// TwinCAT 3 PLC project lamp_motion
// Title: tmo_lamp_motion
// Company: SLAC
// ProjectVersion: 0.0.0
// ProgramVersion: 3.1.4022.7
// libraries:
//   LCLS General, * (SLAC)
//   lcls-twincat-motion, * (SLAC)
//   Tc2_MC2, * (Beckhoff Automation GmbH)
//   Tc2_Standard, * (Beckhoff Automation GmbH)
//   Tc2_System, * (Beckhoff Automation GmbH)
//   Tc2_Utilities, * (Beckhoff Automation GmbH)
//   Tc3_Module, * (Beckhoff Automation GmbH)
// project tree:
//   GVLs/ GVL_PLC_Interfaces.TcGVL
//   / PlcTask.TcTTO
//   POUs/ Main.TcPOU
// real-time tasks:
//   TASK PlcTask: cycle T#9ms, priority 20, ADS port 350
// motion (NC):
//   TASK NC-Task 1 SAF: cycle T#2ms, priority 4, ADS port 501
//   TASK NC-Task 1 SVB: cycle T#10ms, priority 8, ADS port 511
//   AXIS GasJetX (id 1)
//     Dynamic: Acceleration=2, Deceleration=2, DelayTime=0.008
//     Velo: SlowManual=0.5, FastManual=1, Maximum=1
//     OtherSettings: AllowMotionCmdToSlave=true
//     encoder EncType=19
//       EncPara: ScaleFactorNumerator=5e-05, Inverse=true, MaxCount=#xffffffff
//         SoftEndMinControl: Range=-2
//         SoftEndMaxControl: Range=2
//         Inc: RefSoftSyncMask=#x0000ffff
//     drive DrvType=24
//       DrvPara: Inverse=true
//         Analog: VeloReferenz=12.7, ScaleFactorActTorque=0.1
//         TimeComp: TaskDelayCycles=1
//     controller CtrType=1
//       CtrPara: PriorControlFactor=1
//         PosDiffControl: Range=0.8
//         Observer: BandWidth=20
//   AXIS GasJetY (id 2)
//     Dynamic: Acceleration=2, Deceleration=2, DelayTime=0.008
//     Velo: RefSearch=1, RefSync=1, SlowManual=0.5, FastManual=1, Maximum=8
//     OtherSettings: AllowMotionCmdToSlave=true
//     encoder EncType=19
//       EncPara: ScaleFactorNumerator=5e-05, MaxCount=#xffffffff
//         SoftEndMaxControl: Enable=true, Range=735
//         Inc: RefSoftSyncMask=#x0000ffff
//     drive DrvType=24
//       Analog: VeloReferenz=10, ScaleFactorActTorque=0.1
//       TimeComp: TaskDelayCycles=1
//     controller CtrType=1
//       CtrPara: PriorControlFactor=1
//         PosDiffControl: Range=0.8
//         PID: PosKp=2
//         Observer: BandWidth=20
//   AXIS GasJetZ (id 3)
//     Dynamic: AccelerationMaximum=130, DecelerationMaximum=130, Acceleration=3.01464, Deceleration=3.01464, Jerk=17.8197, DelayTime=0.008
//     Velo: SlowManual=0.5, FastManual=1, Maximum=1
//     TargetPosControl: Range=0.01
//     OtherSettings: AllowMotionCmdToSlave=true
//     encoder EncType=29
//       EncPara: ScaleFactorNumerator=5e-05, MaxCount=#xffffffff
//         Inc: RefSoftSyncMask=#x0000ffff
//     drive DrvType=24
//       DrvPara: Inverse=true
//         Analog: VeloReferenz=12.7, ScaleFactorActTorque=0.1
//         TimeComp: TaskDelayCycles=1
//     controller CtrType=1
//       CtrPara: PriorControlFactor=1
//         PosDiffControl: Range=0.1, Time=0.1
//         Observer: BandWidth=20
//   AXIS GasNeedleX (id 4)
//     Dynamic: Acceleration=0.5, Deceleration=2, DelayTime=0.008
//     Velo: SlowManual=0.5, FastManual=1, Maximum=1
//     PositionAreaControl: Range=0.005
//     OtherSettings: AllowMotionCmdToSlave=true
//     encoder EncType=29
//       EncPara: ScaleFactorNumerator=5e-05, Offset=-214613, MaxCount=#xffffffff
//         SoftEndMinControl: Enable=true, Range=19
//         SoftEndMaxControl: Enable=true, Range=39.5
//         Inc: RefSoftSyncMask=#x0000ffff
//     drive DrvType=24
//       Analog: VeloReferenz=10, ScaleFactorActTorque=0.1
//       TimeComp: TaskDelayCycles=1
//     controller CtrType=1
//       CtrPara: PriorControlFactor=1
//         PosDiffControl: Range=0.5
//         PID: PosKp=2
//         Observer: BandWidth=20
//   AXIS GasNeedleY (id 5)
//     Dynamic: Acceleration=2, Deceleration=2, DelayTime=0.008
//     Velo: SlowManual=0.5, FastManual=1, Maximum=1
//     PositionAreaControl: Range=0.5
//     TargetPosControl: Range=0.001, Time=0.2
//     OtherSettings: AllowMotionCmdToSlave=true
//     encoder EncType=19
//       EncPara: ScaleFactorNumerator=5e-05, MaxCount=#xffffffff
//         Inc: RefSoftSyncMask=#x0000ffff
//     drive DrvType=24
//       Analog: VeloReferenz=13, ScaleFactorActTorque=0.1
//       TimeComp: TaskDelayCycles=1
//     controller CtrType=1
//       CtrPara: PriorControlFactor=1
//         PosDiffControl: Range=0.5
//         PID: PosKp=5
//         Observer: BandWidth=20
//   AXIS GasNeedleZ (id 6)
//     Dynamic: Acceleration=2, Deceleration=2, DelayTime=0.008
//     Velo: SlowManual=0.5, FastManual=1, Maximum=1
//     PositionAreaControl: Range=0.005
//     TargetPosControl: Range=0.5
//     OtherSettings: AllowMotionCmdToSlave=true
//     encoder EncType=19
//       EncPara: ScaleFactorNumerator=5e-05, Inverse=true, MaxCount=#xffffffff
//         SoftEndMinControl: Enable=true, Range=-50
//         SoftEndMaxControl: Enable=true, Range=-25
//         Inc: RefSoftSyncMask=#x0000ffff
//     drive DrvType=24
//       Analog: VeloReferenz=10.5, ScaleFactorActTorque=0.1
//       TimeComp: TaskDelayCycles=1
//     controller CtrType=1
//       CtrPara: PriorControlFactor=1
//         PosDiffControl: Range=0.5
//         Observer: BandWidth=20
//   AXIS SamplePaddleX (id 7)
//     Dynamic: Acceleration=2, Deceleration=2, DelayTime=0.008
//     Velo: Maximum=1
//     TargetPosControl: Range=0.001, Time=0.1
//     OtherSettings: AllowMotionCmdToSlave=true
//     encoder EncType=4
//       EncPara: ScaleFactorNumerator=1e-05, Inverse=true, MaxCount=#xffffffff
//         SoftEndMinControl: Range=-39
//         Inc: RefSoftSyncMask=#x0000ffff
//     drive DrvType=24
//       DrvPara: Inverse=true
//         Analog: VeloReferenz=10, ScaleFactorActTorque=0.1
//         TimeComp: TaskDelayCycles=1
//     controller CtrType=2
//       CtrPara: PriorControlFactor=1
//         PosDiffControl: Range=1
//         PID: PosKp=20, PosExtKp=50, DeadBandPosition=0.0005
//         Observer: BandWidth=20
//   AXIS SamplePaddleY (id 8)
//     Dynamic: Acceleration=2, Deceleration=2, DelayTime=0.008
//     Velo: Maximum=1
//     TargetPosControl: Range=0.001, Time=0.1
//     OtherSettings: AllowMotionCmdToSlave=true
//     encoder EncType=4
//       EncPara: ScaleFactorNumerator=2e-05, Inverse=true, MaxCount=#xffffffff
//         SoftEndMinControl: Range=-10
//         SoftEndMaxControl: Range=10
//         Inc: RefSoftSyncMask=#x0000ffff
//     drive DrvType=24
//       DrvPara: Inverse=true
//         Analog: VeloReferenz=5, ScaleFactorActTorque=0.1
//         TimeComp: TaskDelayCycles=1
//     controller CtrType=2
//       CtrPara: PriorControlFactor=1
//         PosDiffControl: Range=0.5
//         PID: PosKp=20, PosExtKp=50, DeadBandPosition=0.0005
//         Observer: BandWidth=20
//   AXIS SamplePaddleZ (id 9)
//     Dynamic: Acceleration=2, Deceleration=2, DelayTime=0.008
//     Velo: Maximum=1
//     TargetPosControl: Range=0.001, Time=0.1
//     OtherSettings: AllowMotionCmdToSlave=true
//     encoder EncType=4
//       EncPara: ScaleFactorNumerator=1e-05, Inverse=true, MaxCount=#xffffffff
//         Inc: RefSoftSyncMask=#x0000ffff
//     drive DrvType=24
//       DrvPara: Inverse=true
//         Analog: VeloReferenz=10, ScaleFactorActTorque=0.1
//         TimeComp: TaskDelayCycles=1
//     controller CtrType=2
//       CtrPara: PriorControlFactor=1
//         PosDiffControl: Range=1
//         PID: PosKp=20, PosExtKp=50, DeadBandPosition=0.0005
//         Observer: BandWidth=20
//   AXIS FlowCellX (id 10)
//     Dynamic: Acceleration=2, Deceleration=2
//     Velo: Maximum=1
//     OtherSettings: AllowMotionCmdToSlave=true
//     encoder EncType=1
//       EncPara: ScaleFactorNumerator=9.375e-05, ScaleFactorDenominator=1.2
//         Inc: RefSoftSyncMask=#x0000ffff
//     drive DrvType=5
//       Analog: VeloReferenz=10, ScaleFactorActTorque=0.1
//       TimeComp: TaskDelayCycles=1
//     controller CtrType=1
//       CtrPara: PriorControlFactor=1
//         PosDiffControl: Range=0.5
//         Observer: BandWidth=20
//   AXIS FlowCellY (id 11)
//     Dynamic: Acceleration=2, Deceleration=2
//     Velo: Maximum=1
//     OtherSettings: AllowMotionCmdToSlave=true
//     encoder EncType=1
//       EncPara: ScaleFactorNumerator=7.8125e-05, ScaleFactorDenominator=0.8
//         Inc: RefSoftSyncMask=#x0000ffff
//     drive DrvType=5
//       Analog: VeloReferenz=12.5, ScaleFactorActTorque=0.1
//       TimeComp: TaskDelayCycles=1
//     controller CtrType=1
//       CtrPara: PriorControlFactor=1
//         PosDiffControl: Range=0.5
//         Observer: BandWidth=20
//   AXIS FlowCellZ (id 12)
//     Dynamic: Acceleration=2, Deceleration=2
//     Velo: Maximum=1
//     OtherSettings: AllowMotionCmdToSlave=true
//     encoder EncType=1
//       EncPara: ScaleFactorNumerator=7.8125e-05
//         Inc: RefSoftSyncMask=#x0000ffff
//     drive DrvType=5
//       Analog: VeloReferenz=10, ScaleFactorActTorque=0.1
//       TimeComp: TaskDelayCycles=1
//     controller CtrType=1
//       CtrPara: PriorControlFactor=1
//         PosDiffControl: Range=0.5
//         Observer: BandWidth=20
//   AXIS FlowCellTheta (id 13)
//     General: UnitName=Degree
//     Velo: Maximum=10
//     OtherSettings: AllowMotionCmdToSlave=true
//     encoder EncType=1
//       EncPara: ScaleFactorNumerator=0.0003125
//         Inc: RefSoftSyncMask=#x0000ffff
//     drive DrvType=5
//       Analog: VeloReferenz=40, ScaleFactorActTorque=0.1
//       TimeComp: TaskDelayCycles=1
//     controller CtrType=2
//       CtrPara: PriorControlFactor=1
//         PosDiffControl: Range=0.5
//         Observer: BandWidth=20
//   AXIS TIXELX (id 14)
//     Dynamic: Acceleration=2, Deceleration=2, DelayTime=0.008
//     Velo: Maximum=1
//     OtherSettings: AllowMotionCmdToSlave=true
//     encoder EncType=4
//       EncPara: ScaleFactorNumerator=3.90625e-05, Inverse=true, MaxCount=#x0000ffff
//         SoftEndMinControl: Range=-2
//         SoftEndMaxControl: Range=2
//         Inc: RefSoftSyncMask=#x0000ffff
//     drive DrvType=24
//       DrvPara: Inverse=true
//         Analog: VeloReferenz=5, ScaleFactorActTorque=0.1
//         TimeComp: TaskDelayCycles=1
//     controller CtrType=1
//       CtrPara: PriorControlFactor=1
//         PosDiffControl: Range=0.5
//         Observer: BandWidth=20
//   AXIS TIXELY (id 15)
//     Dynamic: Acceleration=2, Deceleration=2, DelayTime=0.008
//     Velo: Maximum=1
//     OtherSettings: AllowMotionCmdToSlave=true
//     encoder EncType=4
//       EncPara: ScaleFactorNumerator=3.90625e-05, Inverse=true, MaxCount=#x0000ffff
//         SoftEndMinControl: Range=-2
//         SoftEndMaxControl: Range=2
//         Inc: RefSoftSyncMask=#x0000ffff
//     drive DrvType=24
//       DrvPara: Inverse=true
//         Analog: VeloReferenz=5, ScaleFactorActTorque=0.1
//         TimeComp: TaskDelayCycles=1
//     controller CtrType=1
//       CtrPara: PriorControlFactor=1
//         PosDiffControl: Range=0.5
//         Observer: BandWidth=20
//   AXIS TIXELZ (id 16)
//     Dynamic: Acceleration=2, Deceleration=2, DelayTime=0.008
//     Velo: Maximum=1
//     OtherSettings: AllowMotionCmdToSlave=true
//     encoder EncType=4
//       EncPara: ScaleFactorNumerator=3.90625e-05, Inverse=true, MaxCount=#x0000ffff
//         SoftEndMinControl: Range=-2
//         SoftEndMaxControl: Range=2
//         Inc: RefSoftSyncMask=#x0000ffff
//     drive DrvType=24
//       DrvPara: Inverse=true
//         Analog: VeloReferenz=5, ScaleFactorActTorque=0.1
//         TimeComp: TaskDelayCycles=1
//     controller CtrType=1
//       CtrPara: PriorControlFactor=1
//         PosDiffControl: Range=0.5
//         Observer: BandWidth=20
// I/O:
//   DEVICE PLC Rail (EtherCAT), AmsNetId 0.0.0.0.2.1
//     Power (EK1200) [EK1200-5000 EtherCAT Power supply (2A E-Bus)]
//       PMPS_FFO [EL2202 2Ch. Dig. Output 24V, 0.5A]
//       License (EL6070) [EL6070 1Ch. Licensing-Terminal]
//       LAMP_MOTION_E03_EL6695 [EL6695 EtherCAT Bridge terminal (Primary)]
//       PLC Junction 1 (EK1122) [EK1122 2 port EtherCAT junction]
//         X1 AtmosphereMotion (EK1100) [EK1100 EtherCAT Coupler (2A E-Bus)]
//           GasJetX-EL7041 [EL7041 1Ch. Stepper motor output stage (50V, 5A)]
//           GasJetY-EL7041 [EL7041 1Ch. Stepper motor output stage (50V, 5A)]
//           GasJetY-Brake-EL2004 [EL2004 4Ch. Dig. Output 24V, 0.5A]
//           GasJetZ-EL7041 [EL7041 1Ch. Stepper motor output stage (50V, 5A)]
//           GasNeedleX-EL7041 [EL7041 1Ch. Stepper motor output stage (50V, 5A)]
//           GasNeedleY-EL7041 [EL7041 1Ch. Stepper motor output stage (50V, 5A)]
//           GasNeedleZ-EL7041 [EL7041 1Ch. Stepper motor output stage (50V, 5A)]
//           FlowCellTheta-EL7041 [EL7041 1Ch. Stepper motor output stage (50V, 5A)]
//           GasJetXY-EL5042 [EL5042 2Ch. BiSS-C Encoder]
//           GasJetZGasNeedleX-EL5042 [EL5042 2Ch. BiSS-C Encoder]
//           GasNeedleYZ-EL5042 [EL5042 2Ch. BiSS-C Encoder]
//           AtmosphereMotion-EK1110 [EK1110 EtherCAT extension]
//         X1 VacuumMotion (EK1100) [EK1100 EtherCAT Coupler (2A E-Bus)]
//           SamplePaddleX-EL7041 [EL7041 1Ch. Stepper motor output stage (50V, 5A)]
//           SamplePaddleXY-EL1084 [EL1084 4Ch. Dig. Input 24V, 3ms, negative]
//           SamplePaddleY-EL7041 [EL7041 1Ch. Stepper motor output stage (50V, 5A)]
//           SamplePaddleX-EL5021 [EL5021 1Ch. Sin/Cos Encoder]
//           SamplePaddleY-EL5021 [EL5021 1Ch. Sin/Cos Encoder]
//           SamplePaddleZ-EL7041 [EL7041 1Ch. Stepper motor output stage (50V, 5A)]
//           SamplePaddleZ-EL1084 [EL1084 4Ch. Dig. Input 24V, 3ms, negative]
//           SamplePaddleZ-EL5021 [EL5021 1Ch. Sin/Cos Encoder]
//           Term 56 (EL9410) [EL9410 E-Bus Power Supplier  (Diagnostics)]
//           Term 57 (EL7041) [EL7041 1Ch. Stepper motor output stage (50V, 5A)]
//           Term 58 (EL5021) [EL5021 1K. Sin/Cos Encoder]
//           Term 59 (EL1084) [EL1084 4Ch. Dig. Input 24V, 3ms, negative]
//           Term 60 (EL7041) [EL7041 1Ch. Stepper motor output stage (50V, 5A)] (disabled)
//           Term 61 (EL5021) [EL5021 1Ch. Sin/Cos Encoder]
//           Term 69 (EL9011) [EL9011 End Terminal]
//         TIXEL (EK1100) [EK1100 EtherCAT Coupler (2A E-Bus)]
//           TIXELX-EL7041 [EL7041 1Ch. Stepper motor output stage (50V, 5A)]
//           TIXELXY_ENC-EL5042 [EL5042 2Ch. BiSS-C Encoder]
//           TIXELY-EL7041 [EL7041 1Ch. Stepper motor output stage (50V, 5A)]
//           TIXELZ-EL7041 [EL7041 1Ch. Stepper motor output stage (50V, 5A)]
//           TIXELZ_ENC-EL5042 [EL5042 2Ch. BiSS-C Encoder]
//           Term 68 (EK1110)
// variable links:
//   (this object) <-> PLC Rail (EtherCAT)/Power (EK1200)/PLC Junction 1 (EK1122)/X1 AtmosphereMotion (EK1100)/GasJetX-EL7041
//     Drive/Inputs/In/nState1 @bit 3 <-> STM Status/Status/Error
//     Drive/Inputs/In/nState1 @bit 5 <-> STM Status/Status/Moving negative
//     Drive/Inputs/In/nState1 @bit 4 <-> STM Status/Status/Moving positive
//     Drive/Inputs/In/nState1 @bit 1 <-> STM Status/Status/Ready
//     Drive/Inputs/In/nState1 <-> STM Status/Status/Ready to enable
//     Drive/Inputs/In/nState1 @bit 6 <-> STM Status/Status/Torque reduced
//     Drive/Inputs/In/nState1 @bit 2 <-> STM Status/Status/Warning
//     Drive/Inputs/In/nState2 @bit 3 <-> STM Status/Status/Digital input 1
//     Drive/Inputs/In/nState2 @bit 4 <-> STM Status/Status/Digital input 2
//     Drive/Inputs/In/nState2 @bit 5 <-> STM Status/Status/Sync error
//     Drive/Inputs/In/nState2 @bit 7 <-> STM Status/Status/TxPDO Toggle
//     Drive/Inputs/In/nState4 @bit 1 <-> WcState/InputToggle
//     Drive/Inputs/In/nState4 <-> WcState/WcState
//     Drive/Outputs/Out/nCtrl1 <-> STM Control/Control/Enable
//     Drive/Outputs/Out/nCtrl1 @bit 2 <-> STM Control/Control/Reduce torque
//     Drive/Outputs/Out/nCtrl1 @bit 1 <-> STM Control/Control/Reset
//     Drive/Outputs/Out/nDataOut2[0] <-> STM Velocity/Velocity
//   (this object) <-> PLC Rail (EtherCAT)/Power (EK1200)/PLC Junction 1 (EK1122)/X1 AtmosphereMotion (EK1100)/GasJetXY-EL5042
//     Enc/Inputs/In/nDataIn1 <-> FB Inputs Channel 1 compact/Position
//     Enc/Inputs/In/nDataIn1 <-> FB Inputs Channel 2 compact/Position
//     Enc/Inputs/In/nState1 @bit 1 <-> FB Inputs Channel 1 compact/Status/Error
//     Enc/Inputs/In/nState1 @bit 1 <-> FB Inputs Channel 2 compact/Status/Error
//     Enc/Inputs/In/nState1 @bit 2 <-> FB Inputs Channel 1 compact/Status/Ready
//     Enc/Inputs/In/nState1 @bit 2 <-> FB Inputs Channel 2 compact/Status/Ready
//     Enc/Inputs/In/nState1 <-> FB Inputs Channel 1 compact/Status/Warning
//     Enc/Inputs/In/nState1 <-> FB Inputs Channel 2 compact/Status/Warning
//     Enc/Inputs/In/nState2 @bit 4 <-> FB Inputs Channel 1 compact/Status/Diag
//     Enc/Inputs/In/nState2 @bit 4 <-> FB Inputs Channel 2 compact/Status/Diag
//     Enc/Inputs/In/nState2 @bit 6 <-> FB Inputs Channel 1 compact/Status/Input cycle counter
//     Enc/Inputs/In/nState2 @bit 6 <-> FB Inputs Channel 2 compact/Status/Input cycle counter
//     Enc/Inputs/In/nState2 @bit 5 <-> FB Inputs Channel 1 compact/Status/TxPDO State
//     Enc/Inputs/In/nState2 @bit 5 <-> FB Inputs Channel 2 compact/Status/TxPDO State
//     Enc/Inputs/In/nState4 @bit 1 <-> WcState/InputToggle
//     Enc/Inputs/In/nState4 <-> WcState/WcState
//   (this object) <-> PLC Rail (EtherCAT)/Power (EK1200)/PLC Junction 1 (EK1122)/X1 AtmosphereMotion (EK1100)/GasJetY-EL7041
//     Drive/Inputs/In/nState1 @bit 3 <-> STM Status/Status/Error
//     Drive/Inputs/In/nState1 @bit 5 <-> STM Status/Status/Moving negative
//     Drive/Inputs/In/nState1 @bit 4 <-> STM Status/Status/Moving positive
//     Drive/Inputs/In/nState1 @bit 1 <-> STM Status/Status/Ready
//     Drive/Inputs/In/nState1 <-> STM Status/Status/Ready to enable
//     Drive/Inputs/In/nState1 @bit 6 <-> STM Status/Status/Torque reduced
//     Drive/Inputs/In/nState1 @bit 2 <-> STM Status/Status/Warning
//     Drive/Inputs/In/nState2 @bit 3 <-> STM Status/Status/Digital input 1
//     Drive/Inputs/In/nState2 @bit 4 <-> STM Status/Status/Digital input 2
//     Drive/Inputs/In/nState2 @bit 5 <-> STM Status/Status/Sync error
//     Drive/Inputs/In/nState2 @bit 7 <-> STM Status/Status/TxPDO Toggle
//     Drive/Inputs/In/nState4 @bit 1 <-> WcState/InputToggle
//     Drive/Inputs/In/nState4 <-> WcState/WcState
//     Drive/Outputs/Out/nCtrl1 <-> STM Control/Control/Enable
//     Drive/Outputs/Out/nCtrl1 @bit 2 <-> STM Control/Control/Reduce torque
//     Drive/Outputs/Out/nCtrl1 @bit 1 <-> STM Control/Control/Reset
//     Drive/Outputs/Out/nDataOut2[0] <-> STM Velocity/Velocity
//   (this object) <-> PLC Rail (EtherCAT)/Power (EK1200)/PLC Junction 1 (EK1122)/X1 AtmosphereMotion (EK1100)/GasJetZ-EL7041
//     Drive/Inputs/In/nState1 @bit 3 <-> STM Status/Status/Error
//     Drive/Inputs/In/nState1 @bit 5 <-> STM Status/Status/Moving negative
//     Drive/Inputs/In/nState1 @bit 4 <-> STM Status/Status/Moving positive
//     Drive/Inputs/In/nState1 @bit 1 <-> STM Status/Status/Ready
//     Drive/Inputs/In/nState1 <-> STM Status/Status/Ready to enable
//     Drive/Inputs/In/nState1 @bit 6 <-> STM Status/Status/Torque reduced
//     Drive/Inputs/In/nState1 @bit 2 <-> STM Status/Status/Warning
//     Drive/Inputs/In/nState2 @bit 3 <-> STM Status/Status/Digital input 1
//     Drive/Inputs/In/nState2 @bit 4 <-> STM Status/Status/Digital input 2
//     Drive/Inputs/In/nState2 @bit 5 <-> STM Status/Status/Sync error
//     Drive/Inputs/In/nState2 @bit 7 <-> STM Status/Status/TxPDO Toggle
//     Drive/Inputs/In/nState4 @bit 1 <-> WcState/InputToggle
//     Drive/Inputs/In/nState4 <-> WcState/WcState
//     Drive/Outputs/Out/nCtrl1 <-> STM Control/Control/Enable
//     Drive/Outputs/Out/nCtrl1 @bit 2 <-> STM Control/Control/Reduce torque
//     Drive/Outputs/Out/nCtrl1 @bit 1 <-> STM Control/Control/Reset
//     Drive/Outputs/Out/nDataOut2[0] <-> STM Velocity/Velocity
//   (this object) <-> PLC Rail (EtherCAT)/Power (EK1200)/PLC Junction 1 (EK1122)/X1 AtmosphereMotion (EK1100)/GasJetZGasNeedleX-EL5042
//     Enc/Inputs/In/nComState @bit 1 <-> WcState/InputToggle
//     Enc/Inputs/In/nComState <-> WcState/WcState
//     Enc/Inputs/In/nDataIn1 <-> FB Inputs Channel 1/Position
//     Enc/Inputs/In/nDataIn1 <-> FB Inputs Channel 2/Position
//     Enc/Inputs/In/nState1 @bit 12 <-> FB Inputs Channel 1/Status/Diag
//     Enc/Inputs/In/nState1 @bit 12 <-> FB Inputs Channel 2/Status/Diag
//     Enc/Inputs/In/nState1 @bit 1 <-> FB Inputs Channel 1/Status/Error
//     Enc/Inputs/In/nState1 @bit 1 <-> FB Inputs Channel 2/Status/Error
//     Enc/Inputs/In/nState1 @bit 14 <-> FB Inputs Channel 1/Status/Input cycle counter
//     Enc/Inputs/In/nState1 @bit 14 <-> FB Inputs Channel 2/Status/Input cycle counter
//     Enc/Inputs/In/nState1 @bit 2 <-> FB Inputs Channel 1/Status/Ready
//     Enc/Inputs/In/nState1 @bit 2 <-> FB Inputs Channel 2/Status/Ready
//     Enc/Inputs/In/nState1 @bit 13 <-> FB Inputs Channel 1/Status/TxPDO State
//     Enc/Inputs/In/nState1 @bit 13 <-> FB Inputs Channel 2/Status/TxPDO State
//     Enc/Inputs/In/nState1 <-> FB Inputs Channel 1/Status/Warning
//     Enc/Inputs/In/nState1 <-> FB Inputs Channel 2/Status/Warning
//   (this object) <-> PLC Rail (EtherCAT)/Power (EK1200)/PLC Junction 1 (EK1122)/X1 AtmosphereMotion (EK1100)/GasNeedleX-EL7041
//     Drive/Inputs/In/nState1 @bit 3 <-> STM Status/Status/Error
//     Drive/Inputs/In/nState1 @bit 5 <-> STM Status/Status/Moving negative
//     Drive/Inputs/In/nState1 @bit 4 <-> STM Status/Status/Moving positive
//     Drive/Inputs/In/nState1 @bit 1 <-> STM Status/Status/Ready
//     Drive/Inputs/In/nState1 <-> STM Status/Status/Ready to enable
//     Drive/Inputs/In/nState1 @bit 6 <-> STM Status/Status/Torque reduced
//     Drive/Inputs/In/nState1 @bit 2 <-> STM Status/Status/Warning
//     Drive/Inputs/In/nState2 @bit 3 <-> STM Status/Status/Digital input 1
//     Drive/Inputs/In/nState2 @bit 4 <-> STM Status/Status/Digital input 2
//     Drive/Inputs/In/nState2 @bit 5 <-> STM Status/Status/Sync error
//     Drive/Inputs/In/nState2 @bit 7 <-> STM Status/Status/TxPDO Toggle
//     Drive/Inputs/In/nState4 @bit 1 <-> WcState/InputToggle
//     Drive/Inputs/In/nState4 <-> WcState/WcState
//     Drive/Outputs/Out/nCtrl1 <-> STM Control/Control/Enable
//     Drive/Outputs/Out/nCtrl1 @bit 2 <-> STM Control/Control/Reduce torque
//     Drive/Outputs/Out/nCtrl1 @bit 1 <-> STM Control/Control/Reset
//     Drive/Outputs/Out/nDataOut2[0] <-> STM Velocity/Velocity
//   (this object) <-> PLC Rail (EtherCAT)/Power (EK1200)/PLC Junction 1 (EK1122)/X1 AtmosphereMotion (EK1100)/GasNeedleY-EL7041
//     Drive/Inputs/In/nState1 @bit 3 <-> STM Status/Status/Error
//     Drive/Inputs/In/nState1 @bit 5 <-> STM Status/Status/Moving negative
//     Drive/Inputs/In/nState1 @bit 4 <-> STM Status/Status/Moving positive
//     Drive/Inputs/In/nState1 @bit 1 <-> STM Status/Status/Ready
//     Drive/Inputs/In/nState1 <-> STM Status/Status/Ready to enable
//     Drive/Inputs/In/nState1 @bit 6 <-> STM Status/Status/Torque reduced
//     Drive/Inputs/In/nState1 @bit 2 <-> STM Status/Status/Warning
//     Drive/Inputs/In/nState2 @bit 3 <-> STM Status/Status/Digital input 1
//     Drive/Inputs/In/nState2 @bit 4 <-> STM Status/Status/Digital input 2
//     Drive/Inputs/In/nState2 @bit 5 <-> STM Status/Status/Sync error
//     Drive/Inputs/In/nState2 @bit 7 <-> STM Status/Status/TxPDO Toggle
//     Drive/Inputs/In/nState4 @bit 1 <-> WcState/InputToggle
//     Drive/Inputs/In/nState4 <-> WcState/WcState
//     Drive/Outputs/Out/nCtrl1 <-> STM Control/Control/Enable
//     Drive/Outputs/Out/nCtrl1 @bit 2 <-> STM Control/Control/Reduce torque
//     Drive/Outputs/Out/nCtrl1 @bit 1 <-> STM Control/Control/Reset
//     Drive/Outputs/Out/nDataOut2[0] <-> STM Velocity/Velocity
//   (this object) <-> PLC Rail (EtherCAT)/Power (EK1200)/PLC Junction 1 (EK1122)/X1 AtmosphereMotion (EK1100)/GasNeedleYZ-EL5042
//     Enc/Inputs/In/nDataIn1 <-> FB Inputs Channel 1 compact/Position
//     Enc/Inputs/In/nDataIn1 <-> FB Inputs Channel 2 compact/Position
//     Enc/Inputs/In/nState1 @bit 1 <-> FB Inputs Channel 1 compact/Status/Error
//     Enc/Inputs/In/nState1 @bit 1 <-> FB Inputs Channel 2 compact/Status/Error
//     Enc/Inputs/In/nState1 @bit 2 <-> FB Inputs Channel 1 compact/Status/Ready
//     Enc/Inputs/In/nState1 @bit 2 <-> FB Inputs Channel 2 compact/Status/Ready
//     Enc/Inputs/In/nState1 <-> FB Inputs Channel 1 compact/Status/Warning
//     Enc/Inputs/In/nState1 <-> FB Inputs Channel 2 compact/Status/Warning
//     Enc/Inputs/In/nState2 @bit 4 <-> FB Inputs Channel 1 compact/Status/Diag
//     Enc/Inputs/In/nState2 @bit 4 <-> FB Inputs Channel 2 compact/Status/Diag
//     Enc/Inputs/In/nState2 @bit 6 <-> FB Inputs Channel 1 compact/Status/Input cycle counter
//     Enc/Inputs/In/nState2 @bit 6 <-> FB Inputs Channel 2 compact/Status/Input cycle counter
//     Enc/Inputs/In/nState2 @bit 5 <-> FB Inputs Channel 1 compact/Status/TxPDO State
//     Enc/Inputs/In/nState2 @bit 5 <-> FB Inputs Channel 2 compact/Status/TxPDO State
//     Enc/Inputs/In/nState4 @bit 1 <-> WcState/InputToggle
//     Enc/Inputs/In/nState4 <-> WcState/WcState
//   (this object) <-> PLC Rail (EtherCAT)/Power (EK1200)/PLC Junction 1 (EK1122)/X1 AtmosphereMotion (EK1100)/GasNeedleZ-EL7041
//     Drive/Inputs/In/nState1 @bit 3 <-> STM Status/Status/Error
//     Drive/Inputs/In/nState1 @bit 5 <-> STM Status/Status/Moving negative
//     Drive/Inputs/In/nState1 @bit 4 <-> STM Status/Status/Moving positive
//     Drive/Inputs/In/nState1 @bit 1 <-> STM Status/Status/Ready
//     Drive/Inputs/In/nState1 <-> STM Status/Status/Ready to enable
//     Drive/Inputs/In/nState1 @bit 6 <-> STM Status/Status/Torque reduced
//     Drive/Inputs/In/nState1 @bit 2 <-> STM Status/Status/Warning
//     Drive/Inputs/In/nState2 @bit 3 <-> STM Status/Status/Digital input 1
//     Drive/Inputs/In/nState2 @bit 4 <-> STM Status/Status/Digital input 2
//     Drive/Inputs/In/nState2 @bit 5 <-> STM Status/Status/Sync error
//     Drive/Inputs/In/nState2 @bit 7 <-> STM Status/Status/TxPDO Toggle
//     Drive/Inputs/In/nState4 @bit 1 <-> WcState/InputToggle
//     Drive/Inputs/In/nState4 <-> WcState/WcState
//     Drive/Outputs/Out/nCtrl1 <-> STM Control/Control/Enable
//     Drive/Outputs/Out/nCtrl1 @bit 2 <-> STM Control/Control/Reduce torque
//     Drive/Outputs/Out/nCtrl1 @bit 1 <-> STM Control/Control/Reset
//     Drive/Outputs/Out/nDataOut2[0] <-> STM Velocity/Velocity
//   (this object) <-> PLC Rail (EtherCAT)/Power (EK1200)/PLC Junction 1 (EK1122)/X1 VacuumMotion (EK1100)/SamplePaddleX-EL5021
//     Enc/Inputs/In/nDataIn1 <-> ENC Status/Counter value
//     Enc/Inputs/In/nDataIn2 <-> ENC Status/Latch value
//     Enc/Inputs/In/nState1 <-> ENC Status/Status/Latch C valid
//     Enc/Inputs/In/nState1 @bit 2 <-> ENC Status/Status/Set counter done
//     Enc/Inputs/In/nState2 @bit 2 <-> ENC Status/Status/Status of input C
//     Enc/Inputs/In/nState2 @bit 5 <-> ENC Status/Status/Sync error
//     Enc/Inputs/In/nState2 @bit 6 <-> ENC Status/Status/TxPDO State
//     Enc/Inputs/In/nState2 @bit 7 <-> ENC Status/Status/TxPDO Toggle
//     Enc/Inputs/In/nState3 @bit 4 <-> ENC Status/Status/Amplitude error
//     Enc/Inputs/In/nState3 @bit 3 <-> ENC Status/Status/Frequency error
//     Enc/Inputs/In/nState4 @bit 1 <-> WcState/InputToggle
//     Enc/Inputs/In/nState4 <-> WcState/WcState
//     Enc/Outputs/Out/nCtrl1 <-> ENC Control/Control/Enable latch C
//     Enc/Outputs/Out/nCtrl1 @bit 2 <-> ENC Control/Control/Set counter
//     Enc/Outputs/Out/nDataOut1 <-> ENC Control/Set counter value
//   (this object) <-> PLC Rail (EtherCAT)/Power (EK1200)/PLC Junction 1 (EK1122)/X1 VacuumMotion (EK1100)/SamplePaddleX-EL7041
//     Drive/Inputs/In/nState1 @bit 3 <-> STM Status/Status/Error
//     Drive/Inputs/In/nState1 @bit 5 <-> STM Status/Status/Moving negative
//     Drive/Inputs/In/nState1 @bit 4 <-> STM Status/Status/Moving positive
//     Drive/Inputs/In/nState1 @bit 1 <-> STM Status/Status/Ready
//     Drive/Inputs/In/nState1 <-> STM Status/Status/Ready to enable
//     Drive/Inputs/In/nState1 @bit 6 <-> STM Status/Status/Torque reduced
//     Drive/Inputs/In/nState1 @bit 2 <-> STM Status/Status/Warning
//     Drive/Inputs/In/nState2 @bit 3 <-> STM Status/Status/Digital input 1
//     Drive/Inputs/In/nState2 @bit 4 <-> STM Status/Status/Digital input 2
//     Drive/Inputs/In/nState2 @bit 5 <-> STM Status/Status/Sync error
//     Drive/Inputs/In/nState2 @bit 7 <-> STM Status/Status/TxPDO Toggle
//     Drive/Inputs/In/nState4 @bit 1 <-> WcState/InputToggle
//     Drive/Inputs/In/nState4 <-> WcState/WcState
//     Drive/Outputs/Out/nCtrl1 <-> STM Control/Control/Enable
//     Drive/Outputs/Out/nCtrl1 @bit 2 <-> STM Control/Control/Reduce torque
//     Drive/Outputs/Out/nCtrl1 @bit 1 <-> STM Control/Control/Reset
//     Drive/Outputs/Out/nDataOut2[0] <-> STM Velocity/Velocity
//   (this object) <-> PLC Rail (EtherCAT)/Power (EK1200)/PLC Junction 1 (EK1122)/X1 VacuumMotion (EK1100)/SamplePaddleY-EL5021
//     Enc/Inputs/In/nDataIn1 <-> ENC Status/Counter value
//     Enc/Inputs/In/nDataIn2 <-> ENC Status/Latch value
//     Enc/Inputs/In/nState1 <-> ENC Status/Status/Latch C valid
//     Enc/Inputs/In/nState1 @bit 2 <-> ENC Status/Status/Set counter done
//     Enc/Inputs/In/nState2 @bit 2 <-> ENC Status/Status/Status of input C
//     Enc/Inputs/In/nState2 @bit 5 <-> ENC Status/Status/Sync error
//     Enc/Inputs/In/nState2 @bit 6 <-> ENC Status/Status/TxPDO State
//     Enc/Inputs/In/nState2 @bit 7 <-> ENC Status/Status/TxPDO Toggle
//     Enc/Inputs/In/nState3 @bit 4 <-> ENC Status/Status/Amplitude error
//     Enc/Inputs/In/nState3 @bit 3 <-> ENC Status/Status/Frequency error
//     Enc/Inputs/In/nState4 @bit 1 <-> WcState/InputToggle
//     Enc/Inputs/In/nState4 <-> WcState/WcState
//     Enc/Outputs/Out/nCtrl1 <-> ENC Control/Control/Enable latch C
//     Enc/Outputs/Out/nCtrl1 @bit 2 <-> ENC Control/Control/Set counter
//     Enc/Outputs/Out/nDataOut1 <-> ENC Control/Set counter value
//   (this object) <-> PLC Rail (EtherCAT)/Power (EK1200)/PLC Junction 1 (EK1122)/X1 VacuumMotion (EK1100)/SamplePaddleY-EL7041
//     Drive/Inputs/In/nState1 @bit 3 <-> STM Status/Status/Error
//     Drive/Inputs/In/nState1 @bit 5 <-> STM Status/Status/Moving negative
//     Drive/Inputs/In/nState1 @bit 4 <-> STM Status/Status/Moving positive
//     Drive/Inputs/In/nState1 @bit 1 <-> STM Status/Status/Ready
//     Drive/Inputs/In/nState1 <-> STM Status/Status/Ready to enable
//     Drive/Inputs/In/nState1 @bit 6 <-> STM Status/Status/Torque reduced
//     Drive/Inputs/In/nState1 @bit 2 <-> STM Status/Status/Warning
//     Drive/Inputs/In/nState2 @bit 3 <-> STM Status/Status/Digital input 1
//     Drive/Inputs/In/nState2 @bit 4 <-> STM Status/Status/Digital input 2
//     Drive/Inputs/In/nState2 @bit 5 <-> STM Status/Status/Sync error
//     Drive/Inputs/In/nState2 @bit 7 <-> STM Status/Status/TxPDO Toggle
//     Drive/Inputs/In/nState4 @bit 1 <-> WcState/InputToggle
//     Drive/Inputs/In/nState4 <-> WcState/WcState
//     Drive/Outputs/Out/nCtrl1 <-> STM Control/Control/Enable
//     Drive/Outputs/Out/nCtrl1 @bit 2 <-> STM Control/Control/Reduce torque
//     Drive/Outputs/Out/nCtrl1 @bit 1 <-> STM Control/Control/Reset
//     Drive/Outputs/Out/nDataOut2[0] <-> STM Velocity/Velocity
//   (this object) <-> PLC Rail (EtherCAT)/Power (EK1200)/PLC Junction 1 (EK1122)/X1 VacuumMotion (EK1100)/SamplePaddleZ-EL5021
//     Enc/Inputs/In/nDataIn1 <-> ENC Status/Counter value
//     Enc/Inputs/In/nDataIn2 <-> ENC Status/Latch value
//     Enc/Inputs/In/nState1 <-> ENC Status/Status/Latch C valid
//     Enc/Inputs/In/nState1 @bit 2 <-> ENC Status/Status/Set counter done
//     Enc/Inputs/In/nState2 @bit 2 <-> ENC Status/Status/Status of input C
//     Enc/Inputs/In/nState2 @bit 5 <-> ENC Status/Status/Sync error
//     Enc/Inputs/In/nState2 @bit 6 <-> ENC Status/Status/TxPDO State
//     Enc/Inputs/In/nState2 @bit 7 <-> ENC Status/Status/TxPDO Toggle
//     Enc/Inputs/In/nState3 @bit 4 <-> ENC Status/Status/Amplitude error
//     Enc/Inputs/In/nState3 @bit 3 <-> ENC Status/Status/Frequency error
//     Enc/Inputs/In/nState4 @bit 1 <-> WcState/InputToggle
//     Enc/Inputs/In/nState4 <-> WcState/WcState
//     Enc/Outputs/Out/nCtrl1 <-> ENC Control/Control/Enable latch C
//     Enc/Outputs/Out/nCtrl1 @bit 2 <-> ENC Control/Control/Set counter
//     Enc/Outputs/Out/nDataOut1 <-> ENC Control/Set counter value
//   (this object) <-> PLC Rail (EtherCAT)/Power (EK1200)/PLC Junction 1 (EK1122)/X1 VacuumMotion (EK1100)/SamplePaddleZ-EL7041
//     Drive/Inputs/In/nState1 @bit 3 <-> STM Status/Status/Error
//     Drive/Inputs/In/nState1 @bit 5 <-> STM Status/Status/Moving negative
//     Drive/Inputs/In/nState1 @bit 4 <-> STM Status/Status/Moving positive
//     Drive/Inputs/In/nState1 @bit 1 <-> STM Status/Status/Ready
//     Drive/Inputs/In/nState1 <-> STM Status/Status/Ready to enable
//     Drive/Inputs/In/nState1 @bit 6 <-> STM Status/Status/Torque reduced
//     Drive/Inputs/In/nState1 @bit 2 <-> STM Status/Status/Warning
//     Drive/Inputs/In/nState2 @bit 3 <-> STM Status/Status/Digital input 1
//     Drive/Inputs/In/nState2 @bit 4 <-> STM Status/Status/Digital input 2
//     Drive/Inputs/In/nState2 @bit 5 <-> STM Status/Status/Sync error
//     Drive/Inputs/In/nState2 @bit 7 <-> STM Status/Status/TxPDO Toggle
//     Drive/Inputs/In/nState4 @bit 1 <-> WcState/InputToggle
//     Drive/Inputs/In/nState4 <-> WcState/WcState
//     Drive/Outputs/Out/nCtrl1 <-> STM Control/Control/Enable
//     Drive/Outputs/Out/nCtrl1 @bit 2 <-> STM Control/Control/Reduce torque
//     Drive/Outputs/Out/nCtrl1 @bit 1 <-> STM Control/Control/Reset
//     Drive/Outputs/Out/nDataOut2[0] <-> STM Velocity/Velocity
//   (this object) <-> PLC Rail (EtherCAT)/Power (EK1200)/PLC Junction 1 (EK1122)/TIXEL (EK1100)/TIXELX-EL7041
//     Drive/Inputs/In/nState1 @bit 3 <-> STM Status/Status/Error
//     Drive/Inputs/In/nState1 @bit 5 <-> STM Status/Status/Moving negative
//     Drive/Inputs/In/nState1 @bit 4 <-> STM Status/Status/Moving positive
//     Drive/Inputs/In/nState1 @bit 1 <-> STM Status/Status/Ready
//     Drive/Inputs/In/nState1 <-> STM Status/Status/Ready to enable
//     Drive/Inputs/In/nState1 @bit 6 <-> STM Status/Status/Torque reduced
//     Drive/Inputs/In/nState1 @bit 2 <-> STM Status/Status/Warning
//     Drive/Inputs/In/nState2 @bit 3 <-> STM Status/Status/Digital input 1
//     Drive/Inputs/In/nState2 @bit 4 <-> STM Status/Status/Digital input 2
//     Drive/Inputs/In/nState2 @bit 5 <-> STM Status/Status/Sync error
//     Drive/Inputs/In/nState2 @bit 7 <-> STM Status/Status/TxPDO Toggle
//     Drive/Inputs/In/nState4 @bit 1 <-> WcState/InputToggle
//     Drive/Inputs/In/nState4 <-> WcState/WcState
//     Drive/Outputs/Out/nCtrl1 <-> STM Control/Control/Enable
//     Drive/Outputs/Out/nCtrl1 @bit 2 <-> STM Control/Control/Reduce torque
//     Drive/Outputs/Out/nCtrl1 @bit 1 <-> STM Control/Control/Reset
//     Drive/Outputs/Out/nDataOut2[0] <-> STM Velocity/Velocity
//     Enc/Inputs/In/nDataIn1[0] <-> ENC Status compact/Counter value
//     Enc/Inputs/In/nDataIn2[0] <-> ENC Status compact/Latch value
//     Enc/Inputs/In/nState1 @bit 4 <-> ENC Status compact/Status/Counter overflow
//     Enc/Inputs/In/nState1 @bit 3 <-> ENC Status compact/Status/Counter underflow
//     Enc/Inputs/In/nState1 @bit 7 <-> ENC Status compact/Status/Extrapolation stall
//     Enc/Inputs/In/nState1 <-> ENC Status compact/Status/Latch C valid
//     Enc/Inputs/In/nState1 @bit 1 <-> ENC Status compact/Status/Latch extern valid
//     Enc/Inputs/In/nState1 @bit 2 <-> ENC Status compact/Status/Set counter done
//     Enc/Inputs/In/nState2 @bit 4 <-> ENC Status compact/Status/Status of extern latch
//     Enc/Inputs/In/nState2 <-> ENC Status compact/Status/Status of input A
//     Enc/Inputs/In/nState2 @bit 1 <-> ENC Status compact/Status/Status of input B
//     Enc/Inputs/In/nState2 @bit 2 <-> ENC Status compact/Status/Status of input C
//     Enc/Inputs/In/nState2 @bit 5 <-> ENC Status compact/Status/Sync error
//     Enc/Inputs/In/nState2 @bit 7 <-> ENC Status compact/Status/TxPDO Toggle
//     Enc/Inputs/In/nState4 @bit 1 <-> WcState/InputToggle
//     Enc/Inputs/In/nState4 <-> WcState/WcState
//     Enc/Outputs/Out/nCtrl1 <-> ENC Control compact/Control/Enable latch C
//     Enc/Outputs/Out/nCtrl1 @bit 3 <-> ENC Control compact/Control/Enable latch extern on negative edge
//     Enc/Outputs/Out/nCtrl1 @bit 1 <-> ENC Control compact/Control/Enable latch extern on positive edge
//     Enc/Outputs/Out/nCtrl1 @bit 2 <-> ENC Control compact/Control/Set counter
//     Enc/Outputs/Out/nDataOut1[0] <-> ENC Control compact/Set counter value
//   (this object) <-> PLC Rail (EtherCAT)/Power (EK1200)/PLC Junction 1 (EK1122)/TIXEL (EK1100)/TIXELY-EL7041
//     Drive/Inputs/In/nState1 @bit 3 <-> STM Status/Status/Error
//     Drive/Inputs/In/nState1 @bit 5 <-> STM Status/Status/Moving negative
//     Drive/Inputs/In/nState1 @bit 4 <-> STM Status/Status/Moving positive
//     Drive/Inputs/In/nState1 @bit 1 <-> STM Status/Status/Ready
//     Drive/Inputs/In/nState1 <-> STM Status/Status/Ready to enable
//     Drive/Inputs/In/nState1 @bit 6 <-> STM Status/Status/Torque reduced
//     Drive/Inputs/In/nState1 @bit 2 <-> STM Status/Status/Warning
//     Drive/Inputs/In/nState2 @bit 3 <-> STM Status/Status/Digital input 1
//     Drive/Inputs/In/nState2 @bit 4 <-> STM Status/Status/Digital input 2
//     Drive/Inputs/In/nState2 @bit 5 <-> STM Status/Status/Sync error
//     Drive/Inputs/In/nState2 @bit 7 <-> STM Status/Status/TxPDO Toggle
//     Drive/Inputs/In/nState4 @bit 1 <-> WcState/InputToggle
//     Drive/Inputs/In/nState4 <-> WcState/WcState
//     Drive/Outputs/Out/nCtrl1 <-> STM Control/Control/Enable
//     Drive/Outputs/Out/nCtrl1 @bit 2 <-> STM Control/Control/Reduce torque
//     Drive/Outputs/Out/nCtrl1 @bit 1 <-> STM Control/Control/Reset
//     Drive/Outputs/Out/nDataOut2[0] <-> STM Velocity/Velocity
//     Enc/Inputs/In/nDataIn1[0] <-> ENC Status compact/Counter value
//     Enc/Inputs/In/nDataIn2[0] <-> ENC Status compact/Latch value
//     Enc/Inputs/In/nState1 @bit 4 <-> ENC Status compact/Status/Counter overflow
//     Enc/Inputs/In/nState1 @bit 3 <-> ENC Status compact/Status/Counter underflow
//     Enc/Inputs/In/nState1 @bit 7 <-> ENC Status compact/Status/Extrapolation stall
//     Enc/Inputs/In/nState1 <-> ENC Status compact/Status/Latch C valid
//     Enc/Inputs/In/nState1 @bit 1 <-> ENC Status compact/Status/Latch extern valid
//     Enc/Inputs/In/nState1 @bit 2 <-> ENC Status compact/Status/Set counter done
//     Enc/Inputs/In/nState2 @bit 4 <-> ENC Status compact/Status/Status of extern latch
//     Enc/Inputs/In/nState2 <-> ENC Status compact/Status/Status of input A
//     Enc/Inputs/In/nState2 @bit 1 <-> ENC Status compact/Status/Status of input B
//     Enc/Inputs/In/nState2 @bit 2 <-> ENC Status compact/Status/Status of input C
//     Enc/Inputs/In/nState2 @bit 5 <-> ENC Status compact/Status/Sync error
//     Enc/Inputs/In/nState2 @bit 7 <-> ENC Status compact/Status/TxPDO Toggle
//     Enc/Inputs/In/nState4 @bit 1 <-> WcState/InputToggle
//     Enc/Inputs/In/nState4 <-> WcState/WcState
//     Enc/Outputs/Out/nCtrl1 <-> ENC Control compact/Control/Enable latch C
//     Enc/Outputs/Out/nCtrl1 @bit 3 <-> ENC Control compact/Control/Enable latch extern on negative edge
//     Enc/Outputs/Out/nCtrl1 @bit 1 <-> ENC Control compact/Control/Enable latch extern on positive edge
//     Enc/Outputs/Out/nCtrl1 @bit 2 <-> ENC Control compact/Control/Set counter
//     Enc/Outputs/Out/nDataOut1[0] <-> ENC Control compact/Set counter value
//   (this object) <-> PLC Rail (EtherCAT)/Power (EK1200)/PLC Junction 1 (EK1122)/TIXEL (EK1100)/TIXELZ-EL7041
//     Drive/Inputs/In/nState1 @bit 3 <-> STM Status/Status/Error
//     Drive/Inputs/In/nState1 @bit 5 <-> STM Status/Status/Moving negative
//     Drive/Inputs/In/nState1 @bit 4 <-> STM Status/Status/Moving positive
//     Drive/Inputs/In/nState1 @bit 1 <-> STM Status/Status/Ready
//     Drive/Inputs/In/nState1 <-> STM Status/Status/Ready to enable
//     Drive/Inputs/In/nState1 @bit 6 <-> STM Status/Status/Torque reduced
//     Drive/Inputs/In/nState1 @bit 2 <-> STM Status/Status/Warning
//     Drive/Inputs/In/nState2 @bit 3 <-> STM Status/Status/Digital input 1
//     Drive/Inputs/In/nState2 @bit 4 <-> STM Status/Status/Digital input 2
//     Drive/Inputs/In/nState2 @bit 5 <-> STM Status/Status/Sync error
//     Drive/Inputs/In/nState2 @bit 7 <-> STM Status/Status/TxPDO Toggle
//     Drive/Inputs/In/nState4 @bit 1 <-> WcState/InputToggle
//     Drive/Inputs/In/nState4 <-> WcState/WcState
//     Drive/Outputs/Out/nCtrl1 <-> STM Control/Control/Enable
//     Drive/Outputs/Out/nCtrl1 @bit 2 <-> STM Control/Control/Reduce torque
//     Drive/Outputs/Out/nCtrl1 @bit 1 <-> STM Control/Control/Reset
//     Drive/Outputs/Out/nDataOut2[0] <-> STM Velocity/Velocity
//     Enc/Inputs/In/nDataIn1[0] <-> ENC Status compact/Counter value
//     Enc/Inputs/In/nDataIn2[0] <-> ENC Status compact/Latch value
//     Enc/Inputs/In/nState1 @bit 4 <-> ENC Status compact/Status/Counter overflow
//     Enc/Inputs/In/nState1 @bit 3 <-> ENC Status compact/Status/Counter underflow
//     Enc/Inputs/In/nState1 @bit 7 <-> ENC Status compact/Status/Extrapolation stall
//     Enc/Inputs/In/nState1 <-> ENC Status compact/Status/Latch C valid
//     Enc/Inputs/In/nState1 @bit 1 <-> ENC Status compact/Status/Latch extern valid
//     Enc/Inputs/In/nState1 @bit 2 <-> ENC Status compact/Status/Set counter done
//     Enc/Inputs/In/nState2 @bit 4 <-> ENC Status compact/Status/Status of extern latch
//     Enc/Inputs/In/nState2 <-> ENC Status compact/Status/Status of input A
//     Enc/Inputs/In/nState2 @bit 1 <-> ENC Status compact/Status/Status of input B
//     Enc/Inputs/In/nState2 @bit 2 <-> ENC Status compact/Status/Status of input C
//     Enc/Inputs/In/nState2 @bit 5 <-> ENC Status compact/Status/Sync error
//     Enc/Inputs/In/nState2 @bit 7 <-> ENC Status compact/Status/TxPDO Toggle
//     Enc/Inputs/In/nState4 @bit 1 <-> WcState/InputToggle
//     Enc/Inputs/In/nState4 <-> WcState/WcState
//     Enc/Outputs/Out/nCtrl1 <-> ENC Control compact/Control/Enable latch C
//     Enc/Outputs/Out/nCtrl1 @bit 3 <-> ENC Control compact/Control/Enable latch extern on negative edge
//     Enc/Outputs/Out/nCtrl1 @bit 1 <-> ENC Control compact/Control/Enable latch extern on positive edge
//     Enc/Outputs/Out/nCtrl1 @bit 2 <-> ENC Control compact/Control/Set counter
//     Enc/Outputs/Out/nDataOut1[0] <-> ENC Control compact/Set counter value
//   lamp_motion Instance <-> PLC Rail (EtherCAT)/Power (EK1200)/LAMP_MOTION_E03_EL6695
//     PlcTask Inputs/GVL_PLC_Interfaces.xEcatBridge_TxPDO_state <-> SYNC Inputs/TxPDO state
//     PlcTask Inputs/GVL_PLC_Interfaces.xEcatBridge_WcState <-> WcState/WcState
//     PlcTask Inputs/GVL_PLC_Interfaces.xLAMP_GJ_VRC_01_OPEN_LS <-> IO Inputs/LAMP_GJ_VRC_01_OPEN_LS
//     PlcTask Outputs/GVL_PLC_Interfaces.xLAMP_GJY_OUT <-> IO Outputs/LAMP_GJY_OUT
//   lamp_motion Instance <-> PLC Rail (EtherCAT)/Power (EK1200)/PLC Junction 1 (EK1122)/TIXEL (EK1100)/TIXELX-EL7041
//     PlcTask Inputs/Main.M14.bLimitBackwardEnable <-> STM Status/Status/Digital input 2
//     PlcTask Inputs/Main.M14.bLimitForwardEnable <-> STM Status/Status/Digital input 1
//   lamp_motion Instance <-> PLC Rail (EtherCAT)/Power (EK1200)/PLC Junction 1 (EK1122)/TIXEL (EK1100)/TIXELY-EL7041
//     PlcTask Inputs/Main.M15.bLimitBackwardEnable <-> STM Status/Status/Digital input 2
//     PlcTask Inputs/Main.M15.bLimitForwardEnable <-> STM Status/Status/Digital input 1
//   lamp_motion Instance <-> PLC Rail (EtherCAT)/Power (EK1200)/PLC Junction 1 (EK1122)/TIXEL (EK1100)/TIXELZ-EL7041
//     PlcTask Inputs/Main.M16.bLimitBackwardEnable <-> STM Status/Status/Digital input 2
//     PlcTask Inputs/Main.M16.bLimitForwardEnable <-> STM Status/Status/Digital input 1
//   lamp_motion Instance <-> PLC Rail (EtherCAT)/Power (EK1200)/PLC Junction 1 (EK1122)/X1 AtmosphereMotion (EK1100)/GasJetX-EL7041
//     PlcTask Inputs/Main.M1.bLimitBackwardEnable <-> STM Status/Status/Digital input 2
//     PlcTask Inputs/Main.M1.bLimitForwardEnable <-> STM Status/Status/Digital input 1
//   lamp_motion Instance <-> PLC Rail (EtherCAT)/Power (EK1200)/PLC Junction 1 (EK1122)/X1 AtmosphereMotion (EK1100)/GasJetY-Brake-EL2004
//     PlcTask Outputs/Main.M2.bBrakeRelease <-> Channel 1/Output
//   lamp_motion Instance <-> PLC Rail (EtherCAT)/Power (EK1200)/PLC Junction 1 (EK1122)/X1 AtmosphereMotion (EK1100)/GasJetY-EL7041
//     PlcTask Inputs/Main.M2.bLimitBackwardEnable <-> STM Status/Status/Digital input 1
//     PlcTask Inputs/Main.M2.bLimitForwardEnable <-> STM Status/Status/Digital input 2
//   lamp_motion Instance <-> PLC Rail (EtherCAT)/Power (EK1200)/PLC Junction 1 (EK1122)/X1 AtmosphereMotion (EK1100)/GasJetZ-EL7041
//     PlcTask Inputs/Main.M3.bLimitBackwardEnable <-> STM Status/Status/Digital input 1
//     PlcTask Inputs/Main.M3.bLimitForwardEnable <-> STM Status/Status/Digital input 2
//   lamp_motion Instance <-> PLC Rail (EtherCAT)/Power (EK1200)/PLC Junction 1 (EK1122)/X1 AtmosphereMotion (EK1100)/GasJetZGasNeedleX-EL5042
//     PlcTask Inputs/Main.M3.nRawEncoderULINT <-> FB Inputs Channel 1/Position
//   lamp_motion Instance <-> PLC Rail (EtherCAT)/Power (EK1200)/PLC Junction 1 (EK1122)/X1 AtmosphereMotion (EK1100)/GasNeedleX-EL7041
//     PlcTask Inputs/Main.M4.bLimitBackwardEnable <-> STM Status/Status/Digital input 2
//     PlcTask Inputs/Main.M4.bLimitForwardEnable <-> STM Status/Status/Digital input 1
//   lamp_motion Instance <-> PLC Rail (EtherCAT)/Power (EK1200)/PLC Junction 1 (EK1122)/X1 AtmosphereMotion (EK1100)/GasNeedleY-EL7041
//     PlcTask Inputs/Main.M5.bLimitBackwardEnable <-> STM Status/Status/Digital input 2
//     PlcTask Inputs/Main.M5.bLimitForwardEnable <-> STM Status/Status/Digital input 1
//   lamp_motion Instance <-> PLC Rail (EtherCAT)/Power (EK1200)/PLC Junction 1 (EK1122)/X1 AtmosphereMotion (EK1100)/GasNeedleZ-EL7041
//     PlcTask Inputs/Main.M6.bLimitBackwardEnable <-> STM Status/Status/Digital input 1
//     PlcTask Inputs/Main.M6.bLimitForwardEnable <-> STM Status/Status/Digital input 2
//   lamp_motion Instance <-> PLC Rail (EtherCAT)/Power (EK1200)/PLC Junction 1 (EK1122)/X1 VacuumMotion (EK1100)/SamplePaddleXY-EL1084
//     PlcTask Inputs/Main.M7.bLimitBackwardEnable <-> Channel 2/Input
//     PlcTask Inputs/Main.M8.bLimitBackwardEnable <-> Channel 3/Input
//     PlcTask Inputs/Main.M7.bLimitForwardEnable <-> Channel 1/Input
//     PlcTask Inputs/Main.M8.bLimitForwardEnable <-> Channel 4/Input
//   lamp_motion Instance <-> PLC Rail (EtherCAT)/Power (EK1200)/PLC Junction 1 (EK1122)/X1 VacuumMotion (EK1100)/SamplePaddleZ-EL1084
//     PlcTask Inputs/Main.M9.bLimitBackwardEnable <-> Channel 2/Input
//     PlcTask Inputs/Main.M9.bLimitForwardEnable <-> Channel 1/Input
//   lamp_motion Instance <-> NC-Task 1 SAF/Axes/GasJetX
//     PlcTask Inputs/Main.M1.Axis.NcToPlc <-> Outputs/ToPlc
//     PlcTask Outputs/Main.M1.Axis.PlcToNc <-> Inputs/FromPlc
//   lamp_motion Instance <-> NC-Task 1 SAF/Axes/GasJetY
//     PlcTask Inputs/Main.M2.Axis.NcToPlc <-> Outputs/ToPlc
//     PlcTask Outputs/Main.M2.Axis.PlcToNc <-> Inputs/FromPlc
//   lamp_motion Instance <-> NC-Task 1 SAF/Axes/GasJetZ
//     PlcTask Inputs/Main.M3.Axis.NcToPlc <-> Outputs/ToPlc
//     PlcTask Outputs/Main.M3.Axis.PlcToNc <-> Inputs/FromPlc
//   lamp_motion Instance <-> NC-Task 1 SAF/Axes/GasNeedleX
//     PlcTask Inputs/Main.M4.Axis.NcToPlc <-> Outputs/ToPlc
//     PlcTask Outputs/Main.M4.Axis.PlcToNc <-> Inputs/FromPlc
//   lamp_motion Instance <-> NC-Task 1 SAF/Axes/GasNeedleY
//     PlcTask Inputs/Main.M5.Axis.NcToPlc <-> Outputs/ToPlc
//     PlcTask Outputs/Main.M5.Axis.PlcToNc <-> Inputs/FromPlc
//   lamp_motion Instance <-> NC-Task 1 SAF/Axes/GasNeedleZ
//     PlcTask Inputs/Main.M6.Axis.NcToPlc <-> Outputs/ToPlc
//     PlcTask Outputs/Main.M6.Axis.PlcToNc <-> Inputs/FromPlc
//   lamp_motion Instance <-> NC-Task 1 SAF/Axes/SamplePaddleX
//     PlcTask Inputs/Main.M7.Axis.NcToPlc <-> Outputs/ToPlc
//     PlcTask Outputs/Main.M7.Axis.PlcToNc <-> Inputs/FromPlc
//   lamp_motion Instance <-> NC-Task 1 SAF/Axes/SamplePaddleY
//     PlcTask Inputs/Main.M8.Axis.NcToPlc <-> Outputs/ToPlc
//     PlcTask Outputs/Main.M8.Axis.PlcToNc <-> Inputs/FromPlc
//   lamp_motion Instance <-> NC-Task 1 SAF/Axes/SamplePaddleZ
//     PlcTask Inputs/Main.M9.Axis.NcToPlc <-> Outputs/ToPlc
//     PlcTask Outputs/Main.M9.Axis.PlcToNc <-> Inputs/FromPlc
//   lamp_motion Instance <-> NC-Task 1 SAF/Axes/TIXELX
//     PlcTask Inputs/Main.M14.Axis.NcToPlc <-> Outputs/ToPlc
//     PlcTask Outputs/Main.M14.Axis.PlcToNc <-> Inputs/FromPlc
//   lamp_motion Instance <-> NC-Task 1 SAF/Axes/TIXELY
//     PlcTask Inputs/Main.M15.Axis.NcToPlc <-> Outputs/ToPlc
//     PlcTask Outputs/Main.M15.Axis.PlcToNc <-> Inputs/FromPlc
//   lamp_motion Instance <-> NC-Task 1 SAF/Axes/TIXELZ
//     PlcTask Inputs/Main.M16.Axis.NcToPlc <-> Outputs/ToPlc
//     PlcTask Outputs/Main.M16.Axis.PlcToNc <-> Inputs/FromPlc

CONFIGURATION lamp_motion
    RESOURCE PLC ON TwinCAT3
        TASK PlcTask(INTERVAL := T#9ms, PRIORITY := 20);
        PROGRAM Main WITH PlcTask : Main;
    END_RESOURCE
END_CONFIGURATION

// ---- GVLs/GVL_PLC_Interfaces.TcGVL
//{attribute 'qualified_only'}
VAR_GLOBAL
    (*ETHERCAT BRRIDGE COM STATUS*)
    //0: Other side is in OP state, >0: Error
    {attribute 'TcLinkTo' := 'TIIB[LAMP_MOTION_E03_EL6695]^SYNC Inputs^TxPDO state
    '}
    xEcatBridge_TxPDO_state AT %I* :BOOL;

    //0: External device connectd, 1: External device not connected

    {attribute := 'TIIB[LAMP_MOTION_E03_EL6695]^SYNC Inputs^External device not connected
    '}
    xEcatBridge_External_device_not_connected AT %I* : BOOL;

    //0 = Data valid, 1 = Data invalid
    {attribute 'TcLinkTo' := 'TIIB[LAMP_MOTION_E03_EL6695]^WcState^WcState
    '}
    xEcatBridge_WcState AT %I* : BOOL;

    {attribute 'TcLinkTo' := 'TIIB[LAMP_MOTION_E03_EL6695]^IO Inputs^LAMP_GJ_VRC_01_OPEN_LS'}
    xLAMP_GJ_VRC_01_OPEN_LS  AT %I* : BOOL;

    {attribute  'TcLinkTo' := 'TIIB[LAMP_MOTION_E03_EL6695]^IO Outputs^LAMP_GJY_OUT'}
    xLAMP_GJY_OUT AT %Q*: BOOL;

END_VAR

// ---- POUs/Main.TcPOU
PROGRAM Main
VAR
    // Motors
    {attribute 'TcLinkTo' := '.bLimitForwardEnable:=TIIB[GasJetX-EL7041]^STM Status^Status^Digital input 1;
                              .bLimitBackwardEnable:=TIIB[GasJetX-EL7041]^STM Status^Status^Digital input 2'}
 //                             .nRawEncoderULINT     := TIIB[GasJetXY-EL5042]^FB Inputs Channel 1^Position'}
    {attribute 'pytmc' := '
        pv: TMO:LAMP:MMS:01
    '}
    M1		: DUT_MotionStage := (bPowerSelf:=TRUE,
    nEnableMode:=ENUM_StageEnableMode.DURING_MOTION,
//    nEnableMode:=ENUM_StageEnableMode.ALWAYS,
    nHomingMode := ENUM_EpicsHomeCmd.ABSOLUTE_SET); // Gas Jet X

    {attribute 'TcLinkTo' := '.bLimitForwardEnable:=TIIB[GasJetY-EL7041]^STM Status^Status^Digital input 2;
                              .bLimitBackwardEnable:=TIIB[GasJetY-EL7041]^STM Status^Status^Digital input 1;
							  .bBrakeRelease        :=TIIB[GasJetY-Brake-EL2004]^Channel 1^Output;
                              .nRawEncoderULINT     := TIIB[GasJetXY-EL5042]^FB Inputs Channel 2^Position'}
    {attribute 'pytmc' := '
        pv: TMO:LAMP:MMS:02
    '}
    M2		: DUT_MotionStage := (bPowerSelf:=TRUE,
    nEnableMode:=ENUM_StageEnableMode.DURING_MOTION,
//    nEnableMode:=ENUM_StageEnableMode.ALWAYS,
    nHomingMode := ENUM_EpicsHomeCmd.ABSOLUTE_SET); // Gas Jet Y

    {attribute 'TcLinkTo' := '.bLimitForwardEnable:=TIIB[GasJetZ-EL7041]^STM Status^Status^Digital input 2;
                              .bLimitBackwardEnable:=TIIB[GasJetZ-EL7041]^STM Status^Status^Digital input 1;
                              .nRawEncoderULINT     := TIIB[GasJetZGasNeedleX-EL5042]^FB Inputs Channel 1^Position'}
    {attribute 'pytmc' := '
        pv: TMO:LAMP:MMS:03
    '}
    M3		: DUT_MotionStage := (bPowerSelf:=TRUE,
    nEnableMode:=ENUM_StageEnableMode.DURING_MOTION,
//    nEnableMode:=ENUM_StageEnableMode.ALWAYS,
    nHomingMode := ENUM_EpicsHomeCmd.ABSOLUTE_SET); // Gas Jet Z

    {attribute 'TcLinkTo' := '.bLimitForwardEnable:=TIIB[GasNeedleX-EL7041]^STM Status^Status^Digital input 1;
                              .bLimitBackwardEnable:=TIIB[GasNeedleX-EL7041]^STM Status^Status^Digital input 2'}
    {attribute 'pytmc' := '
        pv: TMO:LAMP:MMS:04
    '}
    M4	    : DUT_MotionStage := (bPowerSelf:=TRUE,
    nEnableMode:=ENUM_StageEnableMode.DURING_MOTION,
//    nEnableMode:=ENUM_StageEnableMode.ALWAYS,
    nHomingMode := ENUM_EpicsHomeCmd.ABSOLUTE_SET); // Gas Needle X

    {attribute 'TcLinkTo' := '.bLimitForwardEnable:=TIIB[GasNeedleY-EL7041]^STM Status^Status^Digital input 1;
                              .bLimitBackwardEnable:=TIIB[GasNeedleY-EL7041]^STM Status^Status^Digital input 2'}
    {attribute 'pytmc' := '
        pv: TMO:LAMP:MMS:05
    '}
    M5	    : DUT_MotionStage := (bPowerSelf:=TRUE,
    nEnableMode:=ENUM_StageEnableMode.DURING_MOTION,
//    nEnableMode:=ENUM_StageEnableMode.ALWAYS,
    nHomingMode := ENUM_EpicsHomeCmd.ABSOLUTE_SET); // Gas Needle Y

    {attribute 'TcLinkTo' := '.bLimitForwardEnable:=TIIB[GasNeedleZ-EL7041]^STM Status^Status^Digital input 2;
                              .bLimitBackwardEnable:=TIIB[GasNeedleZ-EL7041]^STM Status^Status^Digital input 1'}
    {attribute 'pytmc' := '
        pv: TMO:LAMP:MMS:06
    '}
    M6	    : DUT_MotionStage := (bPowerSelf:=TRUE,
    nEnableMode:=ENUM_StageEnableMode.DURING_MOTION,
//    nEnableMode:=ENUM_StageEnableMode.ALWAYS,
    nHomingMode := ENUM_EpicsHomeCmd.ABSOLUTE_SET); // Gas Needle Z

    {attribute 'TcLinkTo' := '.bLimitForwardEnable:=TIIB[SamplePaddleXY-EL1084]^Channel 1^Input;
                              .bLimitBackwardEnable:=TIIB[SamplePaddleXY-EL1084]^Channel 2^Input'}
    {attribute 'pytmc' := '
        pv: TMO:LAMP:MMS:07
    '}
    M7  	: DUT_MotionStage := (bPowerSelf:=TRUE); // Sample Paddle X

    {attribute 'TcLinkTo' := '.bLimitForwardEnable:=TIIB[SamplePaddleXY-EL1084]^Channel 4^Input;
                              .bLimitBackwardEnable:=TIIB[SamplePaddleXY-EL1084]^Channel 3^Input'}
    {attribute 'pytmc' := '
        pv: TMO:LAMP:MMS:08
    '}
    M8  	: DUT_MotionStage := (bPowerSelf:=TRUE); // Sample Paddle Y

    {attribute 'TcLinkTo' := '.bLimitForwardEnable:=TIIB[SamplePaddleZ-EL1084]^Channel 1^Input;
                              .bLimitBackwardEnable:=TIIB[SamplePaddleZ-EL1084]^Channel 2^Input'}
    {attribute 'pytmc' := '
        pv: TMO:LAMP:MMS:09
    '}
    M9  	: DUT_MotionStage := (bPowerSelf:=TRUE); // Sample Paddle Z

    // ...//
    // TIXEL
    {attribute 'TcLinkTo' := '	.bLimitForwardEnable:=TIIB[TIXELX-EL7041]^STM Status^Status^Digital input 1;
                                  .bLimitBackwardEnable:=TIIB[TIXELX-EL7041]^STM Status^Status^Digital input 2';
                                .nRawEncoderULINT:=TIIB[TIXELXY_ENC-EL5042]^FB Inputs Channel 1^Position'}
    {attribute 'pytmc' := '
        pv: TMO:LAMP:MMS:14
    '}
    M14		: DUT_MotionStage := (bPowerSelf:=TRUE, nEnableMode:=ENUM_StageEnableMode.DURING_MOTION); // TIXEL X

    {attribute 'TcLinkTo' := '	.bLimitForwardEnable:=TIIB[TIXELY-EL7041]^STM Status^Status^Digital input 1;
                                  .bLimitBackwardEnable:=TIIB[TIXELY-EL7041]^STM Status^Status^Digital input 2';
                                .nRawEncoderULINT:=TIIB[TIXELXY_ENC-EL5042]^FB Inputs Channel 2^Position'}
    {attribute 'pytmc' := '
        pv: TMO:LAMP:MMS:15
    '}
    M15		: DUT_MotionStage := (bPowerSelf:=TRUE, nEnableMode:=ENUM_StageEnableMode.DURING_MOTION); // TIXEL Y

    {attribute 'TcLinkTo' := '	.bLimitForwardEnable:=TIIB[TIXELZ-EL7041]^STM Status^Status^Digital input 1;
                                  .bLimitBackwardEnable:=TIIB[TIXELZ-EL7041]^STM Status^Status^Digital input 2';
                                .nRawEncoderULINT:=TIIB[TIXELZ_ENC-EL5042]^FB Inputs Channel 1^Position'}
    {attribute 'pytmc' := '
        pv: TMO:LAMP:MMS:16
    '}
    M16		: DUT_MotionStage := (bPowerSelf:=TRUE, nEnableMode:=ENUM_StageEnableMode.DURING_MOTION); // TIXEL Z


    fbMotionStageM1	: FB_MotionStage;
    fbMotionStageM2	: FB_MotionStage;
    fbMotionStageM3	: FB_MotionStage;
    fbMotionStageM4	: FB_MotionStage;
    fbMotionStageM5	: FB_MotionStage;
    fbMotionStageM6	: FB_MotionStage;
    fbMotionStageM7	: FB_MotionStage;
    fbMotionStageM8	: FB_MotionStage;
    fbMotionStageM9	: FB_MotionStage;
    //...//
    fbMotionStageM14	: FB_MotionStage;
    fbMotionStageM15	: FB_MotionStage;
    fbMotionStageM16	: FB_MotionStage;
	fbMotionStageM2EPS : FB_EPS;
END_VAR

// Hardware Enable
// Gas Jet
M1.bHardwareEnable	:= TRUE;
M3.bHardwareEnable	:= TRUE;
//Gas needle Y has EPS with lamp-vac
M2.bHardwareEnable	:= TRUE;
fbMotionStageM2EPS(eps:=M2.stEPSForwardEnable);
fbMotionStageM2EPS.setMessage('LAMP_GJ_VRC_01 is close');
fbMotionStageM2EPS.setBit(0,xLAMP_GJ_VRC_01_OPEN_LS);

fbMotionStageM1(stMotionStage:=M1);
fbMotionStageM2(stMotionStage:=M2);
fbMotionStageM3(stMotionStage:=M3);

// Gas Needle
M4.bHardwareEnable	:= TRUE;
M5.bHardwareEnable	:= TRUE;
M6.bHardwareEnable	:= TRUE;

fbMotionStageM4(stMotionStage:=M4);
fbMotionStageM5(stMotionStage:=M5);
fbMotionStageM6(stMotionStage:=M6);

// Sample Paddle
//M7.bHardwareEnable	:= TRUE;
//M8.bHardwareEnable	:= TRUE;
//M9.bHardwareEnable	:= TRUE;

//fbMotionStageM7(stMotionStage:=M7);
//fbMotionStageM8(stMotionStage:=M8);
//fbMotionStageM9(stMotionStage:=M9);

// TIXEL
M14.bHardwareEnable	:= TRUE;
M15.bHardwareEnable	:= TRUE;
M16.bHardwareEnable	:= TRUE;

fbMotionStageM14(stMotionStage:=M14);
fbMotionStageM15(stMotionStage:=M15);
fbMotionStageM16(stMotionStage:=M16);

END_PROGRAM
